TYPE EL2809 :
STRUCT
	bOut1 ,
	bOut2 ,
	bOut3 ,
	bOut4 ,
	bOut5 ,
	bOut6 ,
	bOut7 ,
	bOut8 ,
	bOut9 ,
	bOut10,
	bOut11,
	bOut12,
	bOut13,
	bOut14,
	bOut15,
	bOut16		AT%Q*	:BOOL;
	bWcState	AT%I*	:BOOL;
	uiState		AT%I*	:UINT;
END_STRUCT
END_TYPE

(* stored: Version 1.1.0.1, ProductVersion 3.1.4024.12
   DUT EL2809: Id {f741758b-91ca-4dc2-93c8-efaee7fc3a3d} *)
